/// Saturation. Limits the value to a minimum and maximum value
FUNCTION FUN_SaturationPointer : REAL
VAR_INPUT
	pValue			:POINTER TO REAL;	// Value				
	fMin			:REAL;				// Saturation min value
	fMax			:REAL;				// Saturation max value
END_VAR
VAR_OUTPUT
	bSaturation		:BOOL;
END_VAR

bSaturation := FALSE;
IF pValue^ < fMin THEN
	pValue^ := fMin;
	bSaturation := TRUE;
ELSIF pValue^ > fMax THEN
	pValue^ := fMax;
	bSaturation := TRUE;
END_IF

END_FUNCTION

(* stored: Version 1.1.0.1, ProductVersion 3.1.4024.12
   POU FUN_SaturationPointer: Id {a51d62b0-6c97-46ab-a0b8-a92f8478fa0f}, SpecialFunc None *)
